// TIA Portal V17 export
// export: Created 2022-03-14T21:17:28.0451915Z, ExportSetting WithDefaults, DisplayName Totally Integrated Automation Portal, DisplayVersion V17, DisplayName TIA Portal Openness, DisplayVersion V17, DisplayName TIA Portal Version Control Interface, DisplayVersion V17, DisplayName STEP 7 Professional, DisplayVersion V17, DisplayName STEP 7 Safety, DisplayVersion V17, DisplayName WinCC Advanced / Unified PC, DisplayVersion V17
FUNCTION_BLOCK "EM00_CM02_Conveyor"   // FB31652, LAD
TITLE = EM00_CM02_HornBeacons
{ S7_Optimized_Access := 'TRUE' }
AUTHOR : tech.team.motioncontrol@siemens.com
FAMILY : CPG
VERSION : 1.1
// Support: tech.team.motioncontrol@siemens.com
// stored: AutoNumber true, IsIECCheckEnabled false, IsRetainMemResEnabled false, MemoryReserve 100, SetENOAutomatically false, UDAEnableTagReadback false
   VAR
      statDummy { ExternalAccessible := 'False'; ExternalVisible := 'False'; ExternalWritable := 'False'} : Bool;   // Variable to control a horn
      instConveyor { S7_SetPoint := 'True'} : "Conveyor";
   END_VAR
BEGIN

REGION Network 1: *** Begin the Setpoint Management Information Section ***
END_REGION

REGION Network 2: *** Begin the Logic Section ***
END_REGION

REGION Network 3: Conveyor instance
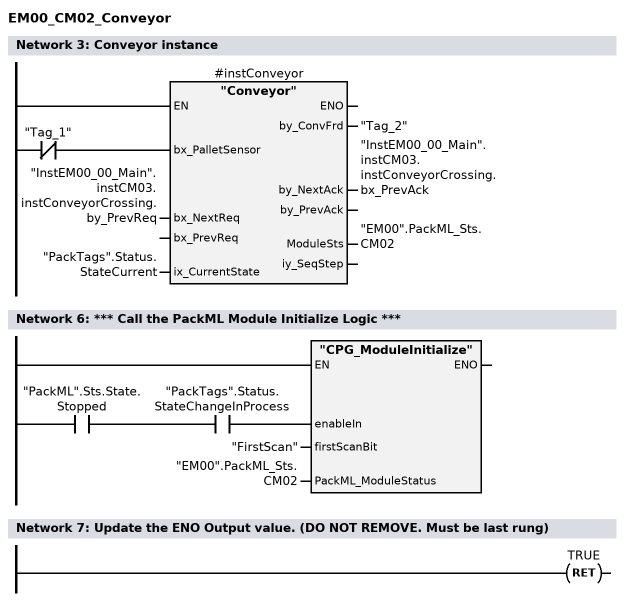
   RUNG wire#powerrail
      #instConveyor(bx_PalletSensor := wire#w1, bx_NextReq := "InstEM00_00_Main".instCM03.instConveyorCrossing.by_PrevReq, bx_PrevReq :=, ix_CurrentState := "PackTags".Status.StateCurrent, by_ConvFrd => "Tag_2", by_NextAck => "InstEM00_00_Main".instCM03.instConveyorCrossing.bx_PrevAck, by_PrevAck =>, ModuleSts => "EM00".PackML_Sts.CM02, iy_SeqStep =>)
   END_RUNG
   RUNG wire#powerrail
      I_Contact( "Tag_1" )
   END_RUNG wire#w1
   // the same network as SCL:
   #instConveyor(bx_PalletSensor := NOT "Tag_1",   // "Conveyor"
                 bx_NextReq := "InstEM00_00_Main".instCM03.instConveyorCrossing.by_PrevReq,
                 ix_CurrentState := "PackTags".Status.StateCurrent,
                 by_ConvFrd => "Tag_2",
                 by_NextAck => "InstEM00_00_Main".instCM03.instConveyorCrossing.bx_PrevAck,
                 ModuleSts => "EM00".PackML_Sts.CM02);
END_REGION

REGION Network 4: *** Begin the Event Information Section ***
END_REGION

REGION Network 5: *** Begin the State Model Status Feedback Section ***
END_REGION

REGION Network 6: *** Call the PackML Module Initialize Logic ***
   RUNG wire#powerrail
      "CPG_ModuleInitialize"(enableIn := wire#w1, firstScanBit := "FirstScan", PackML_ModuleStatus := "EM00".PackML_Sts.CM02)
   END_RUNG
   RUNG wire#powerrail
      Contact( "PackML".Sts.State.Stopped )
      Contact( "PackTags".Status.StateChangeInProcess )
   END_RUNG wire#w1
   // the same network as SCL:
   "CPG_ModuleInitialize"(enableIn := "PackML".Sts.State.Stopped AND "PackTags".Status.StateChangeInProcess,
                          firstScanBit := "FirstScan",
                          PackML_ModuleStatus := "EM00".PackML_Sts.CM02);
END_REGION

REGION Network 7: Update the ENO Output value. (DO NOT REMOVE. Must be last rung)
   RUNG wire#powerrail
      ReturnCoil( TRUE )
   END_RUNG
   // the same network as SCL:
   ENO := TRUE;
   RETURN;
END_REGION
END_FUNCTION_BLOCK
